Staubli VAL3: onF1Event.pgx

program onF1Event()
  local bool l_bYes
  local string l_sMessage
  local string l_sItem
  local num l_nResult
begin
//  // look if the bButton is enable
//  if bButton[0]
//    //
//    //SIMULATION
//    //
//    if !cycleStatus:bCycle and sEvent!=""
//      // load the production page
//      call loadPage("Disk://trajectory/page_simulation",sEvent)
//      // save the moveHold
//      bMoveRelease=false
//    endIf
//  endIf
end
